FUNCTION_BLOCK FB2_Counters
VAR_INPUT
END_VAR
VAR_OUTPUT
END_VAR
VAR
	t_timerHigh : TON;
	t_timerLow : TP;
	b_eenHzTrigger : R_Trig;
	i_productieTimer: DINT;
END_VAR

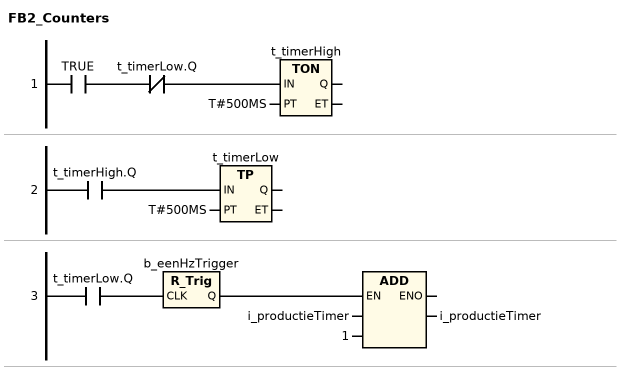
// NETWORK 1
t_timerHigh(IN := TRUE AND NOT t_timerLow.Q, PT := T#500MS); // TON

// NETWORK 2
t_timerLow(IN := t_timerHigh.Q, PT := T#500MS); // TP

// NETWORK 3
b_eenHzTrigger(CLK := t_timerLow.Q); // R_Trig
IF b_eenHzTrigger.Q THEN i_productieTimer := i_productieTimer + 1; END_IF

END_FUNCTION_BLOCK

(* stored: Version 1.1.0.1, ProductVersion 3.1.4024.12
   POU FB2_Counters: Id {37e910bb-9530-4a49-ba25-fc8476665f5e}, SpecialFunc None *)
